// Generic interface for creating clones of objects.
INTERFACE FsI_Cloneable EXTENDS FsI_Unknown

// Returns a clone of the object that exits in dynamic memory.
// Clone must be freed from dynamic memory manually when done.
// A clone is an identical object that occupies a new memory space.
// References from the original object are shared.
METHOD Clone : FsI_Object
VAR_OUTPUT
	e : FsFB_Error;
END_VAR
END_METHOD

END_INTERFACE

(* stored: Version 1.1.0.1, ProductVersion 3.1.4024.4
   Itf FsI_Cloneable: Id {f0cc991c-ad6a-471e-878b-5acab858f1f9}
   Method Clone: Id {27700283-24dd-4d5e-bd76-b85d215190cc} *)
